{attribute 'qualified_only'}
{attribute 'strict'}
TYPE AxisState :
(
	Disabled,
	StandStill,
	Homing,
	DiscreteMotion,
	ContinuousMotion,
	SynchronisedMotion,
	Stopping,
	ErrorStop
) UINT;
END_TYPE

(* stored: Version 1.1.0.1, ProductVersion 3.1.4024.12
   DUT AxisState: Id {77d20cbe-3800-0a98-1db7-2a3caaa54604} *)
